KUKA KRL program: ab_st600_r3_1.src, ab_st600_r3_1.dat

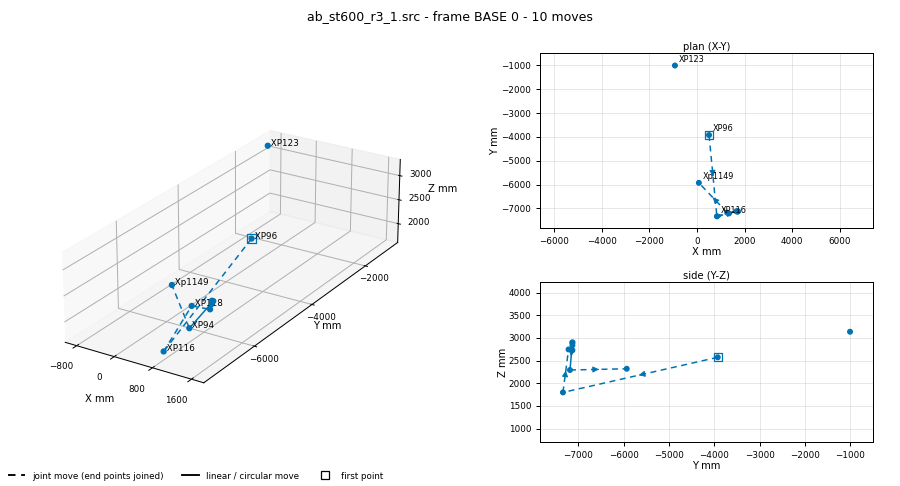
[picture p0: tool path of ab_st600_r3_1.src in frame BASE 0, 10 of 12 moves have a stored position in this frame; points joined in program order, loops and branches not executed]
--- ab_st600_r3_1.src ---
&ACCESS RVO1
&REL 53
&COMMENT Deposita lateral ACTROS
&PARAM DISKPATH = KRC:\R1\Program
DEF AB_ST600_R3_1( )
;FOLD INI
  ;FOLD BASISTECH INI
    GLOBAL INTERRUPT DECL 3 WHEN $STOPMESS==TRUE DO IR_STOPM ( )
    INTERRUPT ON 3
    BAS (#INITMOV,0 )
  ;ENDFOLD (BASISTECH INI)
;FOLD GRIPPERTECH INI
USER_GRP(0,DUMMY,DUMMY,GDEFAULT)
;ENDFOLD (GRIPPERTECH INI)
  ;FOLD USER INI
    ;Make your modifications here

  ;ENDFOLD (USER INI)
;ENDFOLD (INI)

; Caracterização dos meios de produção:
; Versão Atual:
; 12/07/2013 12:00 Name: P13.050-R3 CHANGES: Deposita Lateral Actros
; Gripper (F5 6500 0026 567)

chk_w3_wechs_ok ( )       ; CHECK GRIPPER ACTROS

;FOLD PTP P96 CONT Vel=100 % PDAT90 Tool[3]:Gripper Lateral E.Actros Base[0];%{PE}%R 8.2.20,%MKUKATPBASIS,%CMOVE,%VPTP,%P 1:PTP, 2:P96, 3:C_DIS, 5:100, 7:PDAT90
$BWDSTART=FALSE
PDAT_ACT=PPDAT90
FDAT_ACT=FP96
BAS(#PTP_PARAMS,100)
PTP XP96 C_DIS
;ENDFOLD
;FOLD PTP P116 CONT Vel=100 % PDAT87 Tool[3]:Gripper Lateral E.Actros Base[0];%{PE}%R 8.2.20,%MKUKATPBASIS,%CMOVE,%VPTP,%P 1:PTP, 2:P116, 3:C_DIS, 5:100, 7:PDAT87
$BWDSTART=FALSE
PDAT_ACT=PPDAT87
FDAT_ACT=FP116
BAS(#PTP_PARAMS,100)
PTP XP116 C_DIS
;ENDFOLD

;FOLD Collision.Monitoring_1_On ;%{PE}%MKUKATPUSER
COLLSTOP( 1, 1 ) ;Interrupt-Controlled
;ENDFOLD

;FOLD OUT 3346 'R3 entrega peça Geo' State=TRUE ;%{PE}%R 8.2.20,%MKUKATPBASIS,%COUT,%VOUTX,%P 2:3346, 3:R3 entrega peça Geo, 5:TRUE, 6:
$OUT[3346]=TRUE
;ENDFOLD
;FOLD WAIT FOR ( IN 3346 'Aguarda Lib. entregar peça Geo' );%{PE}%R 8.2.20,%MKUKATPBASIS,%CEXT_WAIT_FOR,%VEXT_WAIT_FOR,%P 2:, 4:, 5:$IN, 6:3346, 7:Aguarda Lib. entregar peça Geo, 9:
WAIT FOR  ( $IN[3346] )
;ENDFOLD
;FOLD OUT 3346 'R3 entrega peça Geo' State=FALSE ;%{PE}%R 8.2.20,%MKUKATPBASIS,%COUT,%VOUTX,%P 2:3346, 3:R3 entrega peça Geo, 5:FALSE, 6:
$OUT[3346]=FALSE
;ENDFOLD
;FOLD OUT 3348 'Fora area GEOBOX' State=FALSE ;%{PE}%R 8.2.20,%MKUKATPBASIS,%COUT,%VOUTX,%P 2:3348, 3:Fora area GEOBOX, 5:FALSE, 6:
$OUT[3348]=FALSE
;ENDFOLD

;FOLD PTP P118 CONT Vel=100 % PDAT120 Tool[3]:Gripper Lateral E.Actros Base[0];%{PE}%R 8.2.20,%MKUKATPBASIS,%CMOVE,%VPTP,%P 1:PTP, 2:P118, 3:C_DIS, 5:100, 7:PDAT120
$BWDSTART=FALSE
PDAT_ACT=PPDAT120
FDAT_ACT=FP118
BAS(#PTP_PARAMS,100)
PTP XP118 C_DIS
;ENDFOLD
;FOLD PTP P120 CONT Vel=100 % PDAT122 Tool[3]:Gripper Lateral E.Actros Base[0];%{PE}%R 8.2.20,%MKUKATPBASIS,%CMOVE,%VPTP,%P 1:PTP, 2:P120, 3:C_DIS, 5:100, 7:PDAT122
$BWDSTART=FALSE
PDAT_ACT=PPDAT122
FDAT_ACT=FP120
BAS(#PTP_PARAMS,100)
PTP XP120 C_DIS
;ENDFOLD
;FOLD PTP p1143 CONT Vel=100 % PDAT110 Tool[3]:Gripper Lateral E.Actros Base[0];%{PE}%R 8.2.20,%MKUKATPBASIS,%CMOVE,%VPTP,%P 1:PTP, 2:p1143, 3:C_DIS, 5:100, 7:PDAT110
$BWDSTART=FALSE
PDAT_ACT=PPDAT110
FDAT_ACT=Fp1143
BAS(#PTP_PARAMS,100)
PTP Xp1143 C_DIS
;ENDFOLD

;FOLD ; PRE ENCAIXE GEOBOX;%{PE}%R 8.2.20,%MKUKATPBASIS,%CCOMMENT,%VNORMAL,%P 2:PRE  ENCAIXE  GEOBOX
;ENDFOLD
;FOLD LIN P85 Vel=0.5 m/s CPDAT41 Tool[3]:Gripper Lateral E.Actros Base[0];%{PE}%R 8.2.20,%MKUKATPBASIS,%CMOVE,%VLIN,%P 1:LIN, 2:P85, 3:, 5:0.5, 7:CPDAT41
$BWDSTART=FALSE
LDAT_ACT=LCPDAT41
FDAT_ACT=FP85
BAS(#CP_PARAMS,0.5)
LIN XP85
;ENDFOLD

;FOLD Collision.Monitoring_AREA_5_Off . ;%{PE}%MKUKATPUSER
COLLSTOP( 11, 2+0 )
;ENDFOLD

;FOLD OUT 3345 'R3 pré encaixe Geo' State=TRUE ;%{PE}%R 8.2.20,%MKUKATPBASIS,%COUT,%VOUTX,%P 2:3345, 3:R3 pré encaixe Geo, 5:TRUE, 6:
$OUT[3345]=TRUE
;ENDFOLD
;FOLD WAIT FOR ( IN 3344 'Aguarda Lib. encaixe na Geo' );%{PE}%R 8.2.20,%MKUKATPBASIS,%CEXT_WAIT_FOR,%VEXT_WAIT_FOR,%P 2:, 4:, 5:$IN, 6:3344, 7:Aguarda Lib. encaixe na Geo, 9:
WAIT FOR  ( $IN[3344] )
;ENDFOLD
;FOLD OUT 3345 'R3 pré encaixe Geo' State=FALSE ;%{PE}%R 8.2.20,%MKUKATPBASIS,%COUT,%VOUTX,%P 2:3345, 3:R3 pré encaixe Geo, 5:FALSE, 6:
$OUT[3345]=FALSE
;ENDFOLD
;FOLD OUT 3344 'R3 solicita lib. sair Geo' State=FALSE ;%{PE}%R 8.2.20,%MKUKATPBASIS,%COUT,%VOUTX,%P 2:3344, 3:R3 solicita lib. sair Geo, 5:FALSE, 6:
$OUT[3344]=FALSE
;ENDFOLD

;FOLD ; PONTO DE DEPOSITO DA PECA NA GEOBOX;%{PE}%R 8.2.20,%MKUKATPBASIS,%CCOMMENT,%VNORMAL,%P 2:PONTO  DE  DEPOSITO  DA  PECA  NA  GEOBOX
;ENDFOLD
;FOLD LIN P112 Vel=0.1 m/s CPDAT45 Tool[3]:Gripper Lateral E.Actros Base[0];%{PE}%R 8.2.20,%MKUKATPBASIS,%CMOVE,%VLIN,%P 1:LIN, 2:P112, 3:, 5:0.1, 7:CPDAT45
$BWDSTART=FALSE
LDAT_ACT=LCPDAT45
FDAT_ACT=FP112
BAS(#CP_PARAMS,0.1)
LIN XP112
;ENDFOLD

;FOLD SET Z2 GRP ACTROS State= GDAT12;%{PE}%R 8.2.1,%MKUKATPGRP,%CGRP,%VGRP,%P 2:2, 4:2, 5:#NO, 6:GDAT12, 8:0, 10:0
H50(GRP,2,2,GGDAT12)
;ENDFOLD
;FOLD SET Z3 GRP ACTROS State=OPN GDAT4;%{PE}%R 8.2.1,%MKUKATPGRP,%CGRP,%VGRP,%P 2:3, 4:1, 5:#NO, 6:GDAT4, 8:0, 10:0
H50(GRP,3,1,GGDAT4)
;ENDFOLD
;FOLD SET Z4.1/2/3/4/5/6/7 ACTROS State=CLO GDAT13;%{PE}%R 8.2.1,%MKUKATPGRP,%CGRP,%VGRP,%P 2:4, 4:2, 5:#NO, 6:GDAT13, 8:0, 10:0
H50(GRP,4,2,GGDAT13)
;ENDFOLD
;FOLD SET Z5 GRP ACTROS State=CLO GDAT14;%{PE}%R 8.2.1,%MKUKATPGRP,%CGRP,%VGRP,%P 2:5, 4:2, 5:#NO, 6:GDAT14, 8:0, 10:0
H50(GRP,5,2,GGDAT14)
;ENDFOLD
chk_w3_grp2_clo()
chk_w3_grp3_opn()
chk_w3_grp4_clo()
chk_w3_grp5_clo()

;FOLD OUT 3344 'R3 solicita lib. sair Geo' State=TRUE ;%{PE}%R 8.2.20,%MKUKATPBASIS,%COUT,%VOUTX,%P 2:3344, 3:R3 solicita lib. sair Geo, 5:TRUE, 6:
$OUT[3344]=TRUE
;ENDFOLD
;FOLD WAIT FOR ( IN 3343 'Aguarda Lib. sair da Geo' );%{PE}%R 8.2.20,%MKUKATPBASIS,%CEXT_WAIT_FOR,%VEXT_WAIT_FOR,%P 2:, 4:, 5:$IN, 6:3343, 7:Aguarda Lib. sair da Geo, 9:
WAIT FOR  ( $IN[3343] )
;ENDFOLD
;FOLD OUT 3344 'R3 solicita lib. sair Geo' State=FALSE ;%{PE}%R 8.2.20,%MKUKATPBASIS,%COUT,%VOUTX,%P 2:3344, 3:R3 solicita lib. sair Geo, 5:FALSE, 6:
$OUT[3344]=FALSE
;ENDFOLD
;FOLD OUT 3343 'R3 entregou peça Geo' State=FALSE ;%{PE}%R 8.2.20,%MKUKATPBASIS,%COUT,%VOUTX,%P 2:3343, 3:R3 entregou peça Geo, 5:FALSE, 6:
$OUT[3343]=FALSE
;ENDFOLD

;FOLD WAIT Time=0.5 sec;%{PE}%R 8.2.20,%MKUKATPBASIS,%CWAIT,%VWAIT,%P 3:0.5
WAIT SEC 0.5
;ENDFOLD
;FOLD OUT 224 'Bloquear MPS' State=FALSE ;%{PE}%R 8.2.20,%MKUKATPBASIS,%COUT,%VOUTX,%P 2:224, 3:Bloquear MPS, 5:FALSE, 6:
$OUT[224]=FALSE
;ENDFOLD
;FOLD OUT 223 'Desbloquear MPS' State=TRUE ;%{PE}%R 8.2.20,%MKUKATPBASIS,%COUT,%VOUTX,%P 2:223, 3:Desbloquear MPS, 5:TRUE, 6:
$OUT[223]=TRUE
;ENDFOLD
;FOLD WAIT FOR ( IN 217 'MPS Destravado' );%{PE}%R 8.2.20,%MKUKATPBASIS,%CEXT_WAIT_FOR,%VEXT_WAIT_FOR,%P 2:, 4:, 5:$IN, 6:217, 7:MPS Destravado, 9:
WAIT FOR  ( $IN[217] )
;ENDFOLD
;FOLD WAIT FOR NOT ( IN 221 'MPS Travado' );%{PE}%R 8.2.20,%MKUKATPBASIS,%CEXT_WAIT_FOR,%VEXT_WAIT_FOR,%P 2:NOT, 4:, 5:$IN, 6:221, 7:MPS Travado, 9:
WAIT FOR  NOT ( $IN[221] )
;ENDFOLD
;FOLD IBUS OFF;%{PE}%R 8.2.20,%MKUKATPBASIS,%CIBUS,%VMAP,%P 2:#OFF, 3:2
$IBUS_OFF=$IBUS_ON
$IBUS_ON=0
;ENDFOLD
;FOLD WAIT Time=0.5 sec;%{PE}%R 8.2.20,%MKUKATPBASIS,%CWAIT,%VWAIT,%P 3:0.5
WAIT SEC 0.5
;ENDFOLD

;FOLD LIN P94 Vel=0.1 m/s CPDAT30 Tool[8]:Tool Changer Base[0];%{PE}%R 8.2.20,%MKUKATPBASIS,%CMOVE,%VLIN,%P 1:LIN, 2:P94, 3:, 5:0.1, 7:CPDAT30
$BWDSTART=FALSE
LDAT_ACT=LCPDAT30
FDAT_ACT=FP94
BAS(#CP_PARAMS,0.1)
LIN XP94
;ENDFOLD

;FOLD WAIT FOR NOT ( IN 219 'Posicao p/ Acoplamento OK' );%{PE}%R 8.2.20,%MKUKATPBASIS,%CEXT_WAIT_FOR,%VEXT_WAIT_FOR,%P 2:NOT, 4:, 5:$IN, 6:219, 7:Posicao p/ Acoplamento OK, 9:
WAIT FOR  NOT ( $IN[219] )
;ENDFOLD
;FOLD OUT 223 'Desbloquear MPS' State=FALSE ;%{PE}%R 8.2.20,%MKUKATPBASIS,%COUT,%VOUTX,%P 2:223, 3:Desbloquear MPS, 5:FALSE, 6:
$OUT[223]=FALSE
;ENDFOLD
;FOLD OUT 3349 'R2 pegou peça' State=FALSE ;%{PE}%R 8.2.20,%MKUKATPBASIS,%COUT,%VOUTX,%P 2:3349, 3:R2 pegou peça, 5:FALSE, 6:
$OUT[3349]=FALSE
;ENDFOLD

;FOLD PTP p1149 CONT Vel=100 % PDAT117 Tool[3]:Gripper Lateral E.Actros Base[0];%{PE}%R 8.2.20,%MKUKATPBASIS,%CMOVE,%VPTP,%P 1:PTP, 2:p1149, 3:C_DIS, 5:100, 7:PDAT117
$BWDSTART=FALSE
PDAT_ACT=PPDAT117
FDAT_ACT=Fp1149
BAS(#PTP_PARAMS,100)
PTP Xp1149 C_DIS
;ENDFOLD

;FOLD OUT 3343 'R3 entregou peça Geo' State=TRUE ;%{PE}%R 8.2.20,%MKUKATPBASIS,%COUT,%VOUTX,%P 2:3343, 3:R3 entregou peça Geo, 5:TRUE, 6:
$OUT[3343]=TRUE
;ENDFOLD
;FOLD OUT 3348 'Fora area GEOBOX' State=TRUE ;%{PE}%R 8.2.20,%MKUKATPBASIS,%COUT,%VOUTX,%P 2:3348, 3:Fora area GEOBOX, 5:TRUE, 6:
$OUT[3348]=TRUE
;ENDFOLD
;FOLD Collision.Monitoring_1_Off . ;%{PE}%MKUKATPUSER
COLLSTOP( 1, 2+0 )
;ENDFOLD

;FOLD PTP P122 CONT Vel=100 % PDAT124 Tool[3]:Gripper Lateral E.Actros Base[0];%{PE}%R 8.2.20,%MKUKATPBASIS,%CMOVE,%VPTP,%P 1:PTP, 2:P122, 3:C_DIS, 5:100, 7:PDAT124
$BWDSTART=FALSE
PDAT_ACT=PPDAT124
FDAT_ACT=FP122
BAS(#PTP_PARAMS,100)
PTP XP122 C_DIS
;ENDFOLD
;FOLD PTP P123 CONT Vel=100 % PDAT125 Tool[3]:Gripper Lateral E.Actros Base[0];%{PE}%R 8.2.20,%MKUKATPBASIS,%CMOVE,%VPTP,%P 1:PTP, 2:P123, 3:C_DIS, 5:100, 7:PDAT125
$BWDSTART=FALSE
PDAT_ACT=PPDAT125
FDAT_ACT=FP123
BAS(#PTP_PARAMS,100)
PTP XP123 C_DIS
;ENDFOLD

;FOLD PTP HOME Vel=100 % PDAT71;%{PE}%R 8.2.20,%MKUKATPBASIS,%CMOVE,%VPTP,%P 1:PTP, 2:HOME, 3:, 5:100, 7:PDAT71
$BWDSTART=FALSE
PDAT_ACT=PPDAT71
FDAT_ACT=FHOME
BAS(#PTP_PARAMS,100)
$H_POS=XHOME
PTP XHOME
;ENDFOLD

END

--- ab_st600_r3_1.dat ---
&ACCESS RVO1
&REL 53
&COMMENT Deposita lateral ACTROS
&PARAM DISKPATH = KRC:\R1\Program
DEFDAT  AB_ST600_R3_1
;FOLD EXTERNAL DECLARATIONS;%{PE}%MKUKATPBASIS,%CEXT,%VCOMMON,%P
;FOLD GRIPPERTECH EXT
EXT  H50 (INT  :IN,INT  :IN,INT  :IN,GRP_TYP  :IN )
;ENDFOLD (GRIPPERTECH EXT)
;FOLD SPOTTECH EXT

;ENDFOLD (SPOTTECH EXT)
;FOLD BASISTECH EXT;%{PE}%MKUKATPBASIS,%CEXT,%VEXT,%P
EXT  BAS (BAS_COMMAND  :IN,REAL  :IN )
DECL INT SUCCESS
;ENDFOLD (BASISTECH EXT)
;FOLD USER EXT;%{E}%MKUKATPUSER,%CEXT,%VEXT,%P
;Make your modifications here

;ENDFOLD (USER EXT)
;ENDFOLD (EXTERNAL DECLARATIONS)INT Segmento

;# ============ START PATH : bh_p13050r3_lta_01 =============
DECL BASIS_SUGG_T LAST_BASIS={POINT1[] "P124                    ",POINT2[] "P124                    ",CP_PARAMS[] "CPDAT0                  ",PTP_PARAMS[] "PDAT126                 ",CONT[] "C_DIS                   ",CP_VEL[] "0.5                     ",PTP_VEL[] "100                     ",SYNC_PARAMS[] "SYNCDAT                 ",SPL_NAME[] "S0                      "}
DECL E6POS XP85={X 1697.74902,Y -7128.24707,Z 2899.57104,A -90.2093124,B 0.0836549923,C -90.0721664,S 6,T 51,E1 5735.10791,E2 0.0,E3 0.0,E4 0.0,E5 0.0,E6 0.0}
DECL FDAT FP85={TOOL_NO 3,BASE_NO 0,IPO_FRAME #BASE,POINT2[] " ",TQ_STATE FALSE}
DECL E6POS XP94={X 1269.62,Y -7181.19922,Z 2293.48193,A -89.9394836,B -74.8758392,C -90.278717,S 2,T 43,E1 5735.10498,E2 0.0,E3 0.0,E4 0.0,E5 0.0,E6 0.0}
DECL FDAT FP94={TOOL_NO 8,BASE_NO 0,IPO_FRAME #BASE,POINT2[] " ",TQ_STATE FALSE}
DECL LDAT LCPDAT30={VEL 2.0,ACC 100.0,APO_DIST 100.0,APO_FAC 50.0,AXIS_VEL 100.0,AXIS_ACC 100.0,ORI_TYP #VAR,CIRC_TYP #BASE,JERK_FAC 50.0,GEAR_JERK 50.0,EXAX_IGN 0}
DECL E6POS XP96={X 506.5961,Y -3923.43311,Z 2573.54297,A -115.927498,B -20.1208,C -108.411903,S 2,T 43,E1 2252.51392,E2 0.0,E3 0.0,E4 0.0,E5 0.0,E6 0.0}
DECL FDAT FP96={TOOL_NO 3,BASE_NO 0,IPO_FRAME #BASE,POINT2[] " ",TQ_STATE FALSE}
DECL PDAT PPDAT71={VEL 100.0,ACC 100.0,APO_DIST 100.0}
DECL E6POS XP112={X 1725.19604,Y -7128.24707,Z 2899.57202,A -90.2092972,B 0.0836288109,C -90.0721512,S 6,T 51,E1 5735.10791,E2 0.0,E3 0.0,E4 0.0,E5 0.0,E6 0.0}
DECL FDAT FP112={TOOL_NO 3,BASE_NO 0,IPO_FRAME #BASE,POINT2[] " ",TQ_STATE FALSE}
DECL E6POS XP116={X 836.222473,Y -7336.04785,Z 1799.34204,A -99.3582687,B -52.5874901,C 63.3023605,S 2,T 43,E1 4431.81299,E2 0.0,E3 0.0,E4 0.0,E5 0.0,E6 0.0}
DECL FDAT FP116={TOOL_NO 1,BASE_NO 0,IPO_FRAME #BASE,POINT2[] " ",TQ_STATE FALSE}
DECL PDAT PPDAT87={VEL 100.0,ACC 100.0,APO_DIST 50.0,APO_MODE #CDIS}
DECL PDAT PPDAT90={VEL 100.0,ACC 100.0,APO_DIST 50.0,APO_MODE #CDIS}
DECL LDAT LCPDAT41={VEL 2.0,ACC 100.0,APO_DIST 100.0,APO_FAC 50.0,AXIS_VEL 100.0,AXIS_ACC 100.0,ORI_TYP #VAR,CIRC_TYP #BASE,JERK_FAC 50.0,GEAR_JERK 50.0,EXAX_IGN 0}
DECL LDAT LCPDAT45={VEL 2.0,ACC 100.0,APO_DIST 100.0,APO_FAC 50.0,AXIS_VEL 100.0,AXIS_ACC 100.0,ORI_TYP #VAR,CIRC_TYP #BASE,JERK_FAC 50.0,GEAR_JERK 50.0,EXAX_IGN 0}
DECL GRP_SUGG_T LAST_GRP={NUMBER[] "2                       ",STATE[] "1                       ",PARAMS[] "GDAT8                   "}
DECL GRP_TYP GGDAT3={G_APO #NO,GRP_TIME 0.200000003,CTRL #OFF,DLY 0,DST 1}
DECL GRP_TYP GGDAT6={G_APO #NO,GRP_TIME 0.200000003,CTRL #OFF,DLY 0,DST 1}
DECL GRP_TYP GGDAT7={G_APO #NO,GRP_TIME 0.200000003,CTRL #OFF,DLY 0,DST 1}
DECL GRP_TYP GGDAT8={G_APO #NO,GRP_TIME 0.200000003,CTRL #OFF,DLY 0,DST 1}
DECL E6POS XP1143={X 1692.72595,Y -7128.14795,Z 2837.646,A -92.6585922,B 0.303313702,C -98.3062286,S 2,T 43,E1 5735.10791,E2 0.0,E3 0.0,E4 0.0,E5 0.0,E6 0.0}
DECL FDAT Fp1143={TOOL_NO 3,BASE_NO 0,IPO_FRAME #BASE,POINT2[] " ",TQ_STATE FALSE}
DECL PDAT PPDAT110={VEL 100.0,ACC 100.0,APO_DIST 50.0,APO_MODE #CDIS}
DECL GRP_TYP GGDAT4={G_APO #NO,GRP_TIME 0.200000003,CTRL #OFF,DLY 0,DST 1}
DECL GRP_TYP GGDAT9={G_APO #NO,GRP_TIME 0.200000003,CTRL #OFF,DLY 0,DST 1}
DECL GRP_TYP GGDAT10={G_APO #NO,GRP_TIME 0.200000003,CTRL #OFF,DLY 0,DST 1}
DECL GRP_TYP GGDAT11={G_APO #NO,GRP_TIME 0.200000003,CTRL #OFF,DLY 0,DST 1}
DECL E6POS XP1149={X 80.1386414,Y -5929.79395,Z 2320.65405,A -66.3707962,B -70.8814774,C -145.585999,S 2,T 43,E1 4458.3291,E2 0.0,E3 0.0,E4 0.0,E5 0.0,E6 0.0}
DECL FDAT Fp1149={TOOL_NO 8,BASE_NO 0,IPO_FRAME #BASE,POINT2[] " ",TQ_STATE FALSE}
DECL PDAT PPDAT117={VEL 100.0,ACC 100.0,APO_DIST 100.0,APO_MODE #CDIS}
DECL GRP_TYP GGDAT12={G_APO #NO,GRP_TIME 0.200000003,CTRL #OFF,DLY 0,DST 1}
DECL GRP_TYP GGDAT13={G_APO #NO,GRP_TIME 0.200000003,CTRL #OFF,DLY 0,DST 1}
DECL GRP_TYP GGDAT14={G_APO #NO,GRP_TIME 0.200000003,CTRL #OFF,DLY 0,DST 1}
DECL E6POS XP118={X 1342.15405,Y -7212.94189,Z 2746.73193,A -95.2293701,B 0.550326228,C -102.8237,S 2,T 43,E1 5570.26318,E2 0.0,E3 0.0,E4 0.0,E5 0.0,E6 0.0}
DECL FDAT FP118={TOOL_NO 3,BASE_NO 0,IPO_FRAME #BASE,POINT2[] " ",TQ_STATE FALSE}
DECL PDAT PPDAT120={VEL 100.0,ACC 100.0,APO_DIST 100.0,APO_MODE #CDIS}
DECL E6POS XP120={X 1659.30103,Y -7127.85889,Z 2728.9209,A -94.5437164,B 1.15150499,C -100.7052,S 2,T 43,E1 5735.10791,E2 0.0,E3 0.0,E4 0.0,E5 0.0,E6 0.0}
DECL FDAT FP120={TOOL_NO 3,BASE_NO 0,IPO_FRAME #BASE,POINT2[] " ",TQ_STATE FALSE}
DECL PDAT PPDAT122={VEL 100.0,ACC 100.0,APO_DIST 50.0,APO_MODE #CDIS}
DECL E6POS XP122={X -4164.69385,Y -2048.65894,Z 1393.39294,A 160.564407,B -77.0369263,C -124.131599,S 2,T 43,E1 376.303314,E2 0.0,E3 0.0,E4 0.0,E5 0.0,E6 0.0}
DECL FDAT FP122={TOOL_NO 2,BASE_NO 2,IPO_FRAME #BASE,POINT2[] " ",TQ_STATE FALSE}
DECL PDAT PPDAT124={VEL 100.0,ACC 100.0,APO_DIST 30.0,APO_MODE #CDIS}
DECL E6POS XP123={X -924.334778,Y -1006.55499,Z 3137.07007,A -39.6929893,B 60.3178787,C 104.575996,S 2,T 10,E1 721.451477,E2 0.0,E3 0.0,E4 0.0,E5 0.0,E6 0.0}
DECL FDAT FP123={TOOL_NO 8,BASE_NO 0,IPO_FRAME #BASE,POINT2[] " ",TQ_STATE FALSE}
DECL PDAT PPDAT125={VEL 100.0,ACC 100.0,APO_DIST 25.0,APO_MODE #CDIS}
ENDDAT
